// TIA Portal V19 export
FUNCTION_BLOCK "SCALE AO"   // FB5, LAD
{ S7_Optimized_Access := 'TRUE' }
// stored: MemoryReserve 100, SetENOAutomatically false
   VAR_INPUT
      "SET RPM" : Real;
      "MIN RPM" : Real;
      "MAX RPM" : Real;
      "MIN HZ" : Int;
      "MAX HZ" : Int;
   END_VAR
   VAR_OUTPUT
      MODBUS : Int;
   END_VAR
   VAR_TEMP
      NOM : Real;
   END_VAR
BEGIN

REGION Network 1
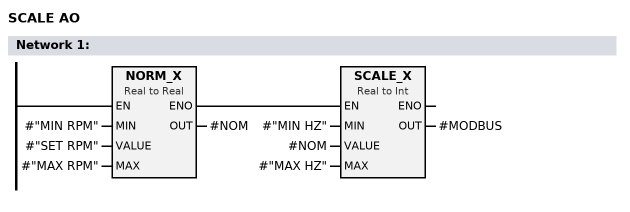
   RUNG wire#powerrail
      { S7_Templates := "[SrcType := Real, DestType := Real]" } Normalize(min := #"MIN RPM", value := #"SET RPM", max := #"MAX RPM", out => #NOM)
      { S7_Templates := "[SrcType := Real, DestType := Int]" } Scale(min := #"MIN HZ", value := #NOM, max := #"MAX HZ", out => #MODBUS)
   END_RUNG
   // the same network as SCL:
   #NOM := NORM_X(MIN := #"MIN RPM", VALUE := #"SET RPM", MAX := #"MAX RPM");
   #MODBUS := SCALE_X(MIN := #"MIN HZ", VALUE := #NOM, MAX := #"MAX HZ");
END_REGION
END_FUNCTION_BLOCK
